FUNCTION_BLOCK GF_Ruehren EXTENDS FB_Basis
VAR_INPUT
	// Instanzieren von Sensoren mit Interfaces
	
	// Instanzieren von Aktoren mit Interfaces
	Ruehrer		:I_Motor1R;
	// Rezeptparamter
END_VAR
VAR_OUTPUT
	
END_VAR
VAR
	
END_VAR

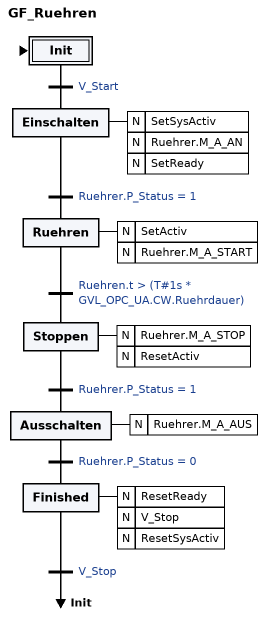
INITIAL_STEP Init:
END_STEP
TRANSITION FROM Init TO Einschalten
    := V_Start;
END_TRANSITION
STEP Einschalten:
    SetSysActiv(N);
    Ruehrer.M_A_AN(N);
    SetReady(N);
END_STEP
TRANSITION FROM Einschalten TO Ruehren
    := Ruehrer.P_Status = 1;
END_TRANSITION
STEP Ruehren:
    SetActiv(N);
    Ruehrer.M_A_START(N);
END_STEP
TRANSITION FROM Ruehren TO Stoppen
    := Ruehren.t > (T#1s * GVL_OPC_UA.CW.Ruehrdauer);
END_TRANSITION
STEP Stoppen:
    Ruehrer.M_A_STOP(N);
    ResetActiv(N);
END_STEP
TRANSITION FROM Stoppen TO Ausschalten
    := Ruehrer.P_Status = 1;
END_TRANSITION
STEP Ausschalten:
    Ruehrer.M_A_AUS(N);
END_STEP
TRANSITION FROM Ausschalten TO Finished
    := Ruehrer.P_Status = 0;
END_TRANSITION
STEP Finished:
    ResetReady(N);
    V_Stop(N);
    ResetSysActiv(N);
END_STEP
TRANSITION FROM Finished TO Init
    := V_Stop;
END_TRANSITION

ACTION ResetActiv:
GVL_OPC_UA.SW.PrimActiv := FALSE;
GVL_OPC_UA.SW.GF5Activ := FALSE;
END_ACTION

ACTION ResetReady:
GVL_OPC_UA.SW.PrimReady := FALSE;
END_ACTION

ACTION ResetSysActiv:
GVL.SysState := 0;
END_ACTION

ACTION SetActiv:
GVL_OPC_UA.SW.PrimActiv := TRUE;
GVL_OPC_UA.SW.GF5Activ := TRUE;
END_ACTION

ACTION SetReady:
GVL_OPC_UA.SW.PrimReady := TRUE;
END_ACTION

ACTION SetSysActiv:
GVL.SysState := 1;
END_ACTION

END_FUNCTION_BLOCK

(* stored: Version 1.1.0.1, ProductVersion 3.1.4024.12
   POU GF_Ruehren: Id {715003b6-7dcf-4be3-a0ad-5b1a6bf337c1}, SpecialFunc None
   Folder 01_Aktionen: Id {cba953e3-74a7-41c0-b82f-a4f3046cdcef}
   Action ResetActiv: Id {d9f6660c-dbad-471b-b9ba-0052e6575729}
   Action ResetReady: Id {131cdfe6-4df2-4bf1-9c25-d5cfb052103d}
   Action ResetSysActiv: Id {b24d2044-49b6-40dd-b3d9-a5655f516cc2}
   Action SetActiv: Id {f891e4ac-89de-4f99-acc4-b9b8774b7345}
   Action SetReady: Id {eb593942-8af3-4940-8f8a-46094f827e62}
   Action SetSysActiv: Id {c96d44b9-9a8d-4b53-8d2a-65042664aad6} *)
